FUNCTION_BLOCK FB_ExampleDeviceGoverner
VAR_INPUT
	stBeamParams	:	ST_BeamParams;
END_VAR
VAR_OUTPUT
	xFault	:	BOOL := TRUE;	
END_VAR
VAR_IN_OUT
	stDevice	:	ST_ExampleDevice;
END_VAR
VAR
	MC_Power: MC_Power;
END_VAR

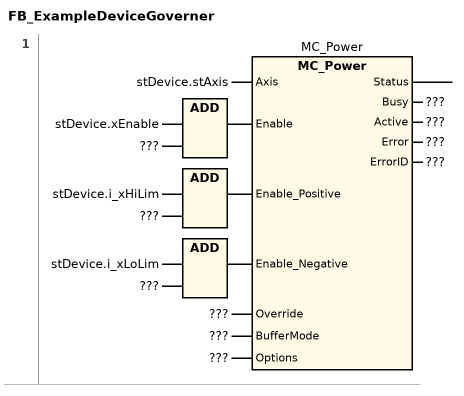
// NETWORK 1
MC_Power(
    Axis := stDevice.stAxis,
    Enable := stDevice.xEnable + ???,
    Enable_Positive := stDevice.i_xHiLim + ???,
    Enable_Negative := stDevice.i_xLoLim + ???);

END_FUNCTION_BLOCK

(* stored: Version 1.1.0.1, ProductVersion 3.1.4022.10
   POU FB_ExampleDeviceGoverner: Id {cd101f41-772b-4bcd-9296-94a4adfc6bb8}, SpecialFunc None *)
